// TIA Portal V17 export
// export: Created 2024-01-30T08:49:14.9649568Z, ExportSetting WithDefaults, DisplayName Totally Integrated Automation Portal, DisplayVersion V17 Update 6, DisplayName TIA Portal Openness, DisplayVersion V17 Update 6, DisplayName TIA Portal Version Control Interface, DisplayVersion V17, DisplayName STEP 7 Professional, DisplayVersion V17 Update 6, DisplayName STEP 7 Safety, DisplayVersion V17 Update 6, DisplayName WinCC Advanced, DisplayVersion V17 Update 6
DATA_BLOCK "B.01813_SIPP_DB"   // DB20
VERSION : 0.1
// stored: AutoNumber true, DBAccessibleFromOPCUA true, DBAccessibleFromWebserver true, InstanceOfName B.01813_SIPP, InstanceOfType FB
"B.01813_SIPP"
   // VAR
   //    SQ_Activation_Time : UDInt;
   //    SQ_Act_time_inH : Real;
   // END_VAR
BEGIN
END_DATA_BLOCK
